PROGRAM MAIN
VAR
	myWord			: WORD := 16#5D7A;
	myResult		: WORD;
	myDword			: DWORD;
	parsedWord		: St_RS232Word;
END_VAR

myResult := SHR(myWord, 3);
myDword  := SHL(myWord, 3);

myDword  := myDword OR 16#F0000000;


parsedWord := FUN_ParseStatusWord(16#1D06);
parsedWord := FUN_ParseStatusWord(16#534C);
parsedWord := FUN_ParseStatusWord(16#C705);

END_PROGRAM

(* stored: Version 1.1.0.1, ProductVersion 3.1.4024.9
   POU MAIN: Id {4101f302-d7e5-462b-a152-df7e24613f81}, SpecialFunc None *)
